// TIA Portal V19 export
VAR_GLOBAL   // PLC tag table "U2Em4"
END_VAR
VAR_GLOBAL CONSTANT   // user constants
   U2EM4_JOB_EXECUTE : DInt := 100;
   U2EM4_JOB_STOPPING : DInt := 200;
   U2EM4_JOB_HOLODING : DInt := 300;
   U2EM4_JOB_UNHOLODING : DInt := 400;
   U2EM4_JOB_RESTING : DInt := 500;
   U2EM4_JOB_STARTING : DInt := 600;
   U2EM4_NO_OF_AXES : USInt := 3;
   U2EM4_JOB_RECOVER : DInt := 700;
END_VAR
